PROGRAM MAIN
VAR
END_VAR

END_PROGRAM

(* stored: Version 1.1.0.1
   POU MAIN: Id {5a41478f-2cb8-4cd8-97b5-4334eb37f2f9} *)
